# EPICS substitutions: IOC/rgt/iocBoot/iocrgt/asynRecord.substitutions
file "$(ASYN)/db/asynRecord.db"
{
pattern
{P        R         PORT    ADDR    OMAX  IMAX}
{rgt:     asyn_1   serial1    0     256  256}
{rgt:     asyn_2   serial2    0     256  256}
{rgt:     asyn_3   serial3    0     256  256}
#{rgt:     asyn_4   serial4    0     256  256}
}
